ORGANIZATION_BLOCK "COMPLETE RESTART"
TITLE =Force glue-scale / Panel LED state to safe idle on every PLC restart
// v0.1 - NEW, per Michou's request (2026-10-06): "need to reset
//   everything when PLC reboots." S7-300 DB "actual values" are
//   battery/cap-backed and survive a power cycle - without this, a
//   reboot mid-recalibration would leave ReCalib_Step stuck mid-sequence
//   while K1/K2 are physically de-energized (CPU zeroes the output
//   process image on every restart, before this OB even runs), and any
//   latched alarms or Panel LED test bits would resume as if nothing
//   happened. Networks below force this repo's own state fields back to
//   a safe idle/off default. Operator setpoints (Fill_Start_SP,
//   Fill_Stop_SP, AlarmLimit_*_SP, PlatformMinWeight_SP,
//   NegativeUnderScore_Value) are deliberately NOT touched here - those
//   are calibration, not state, and must survive a reboot.
//
//   IMPORTANT, CONFIRMED (Michou, 2026-10-06): OB100 already exists on
//   the live PLC project. Michou - paste this file's networks into the
//   END of your existing OB100, do NOT download/replace the whole
//   block - that would silently delete whatever else it already resets
//   for other 410 subsystems. This tracked file only ever represents
//   the networks this repo's own subsystems need, not the real OB100.
//
// v0.2 - per Michou (2026-10-06): "Need a 30 sec delay before
//   restarting after power has resumed ... Need to restart KiloTech
//   Scale too and make sure it is calibrated before operating the
//   pump!" OB100 itself can't block/delay (an OB can't sit and wait -
//   that would trip the scan-time watchdog) - the actual 30s wait and
//   auto-recalibration run in FC155/FB555 (v0.30/v0.4), gated by two
//   new DB105 bits this OB resets every restart: PowerUp_Settled
//   (drives FB555's new 30s startup timer - see FC155's "Timers"
//   network) and Scale_Calibrated (the new pump interlock - see FC155's
//   "Power-up/recalibration interlock" network). Added both resets to
//   the "Glue scale" network below.
//
// v0.3 - reconciled against Michou's own live DB105 refactor
//   (2026-10-07): Reset_Alarms renamed Alarms_Acknowledge - updated the
//   reset below to match. Also added a reset for the new
//   Alarm_PossibleLeak latch (FC155/DB105 v0.20) - missed when that
//   alarm was first added, would have left a possible-leak alarm from
//   before a reboot still latched after it.
VERSION : 0.3


VAR_TEMP
  OB100_EV_CLASS : BYTE ;
  OB100_STRTUP : BYTE ;
  OB100_PRIORITY : BYTE ;
  OB100_OB_NUMBR : BYTE ;
  OB100_RESERVED_1 : BYTE ;
  OB100_RESERVED_2 : BYTE ;
  OB100_STOP : WORD ;
  OB100_STRT_INFO : DWORD ;
  OB100_DATE_TIME : DATE_AND_TIME ;
END_VAR
BEGIN
NETWORK
TITLE =Glue scale - clear latched alarms, HMI trigger pulses, and mid-sequence state (see FC155)

      R     "GLUE SCALE CONTROL DB".Pump_ON;
      R     "GLUE SCALE CONTROL DB".Alarm_Overfill;
      R     "GLUE SCALE CONTROL DB".Alarm_Underfill;
      R     "GLUE SCALE CONTROL DB".Alarm_ScaleFault;
      R     "GLUE SCALE CONTROL DB".ParseError;
      R     "GLUE SCALE CONTROL DB".Pump_ON_Prev;
      R     "GLUE SCALE CONTROL DB".Scale_Powered_On;
      R     "GLUE SCALE CONTROL DB".Alarms_Acknowledge;
      R     "GLUE SCALE CONTROL DB".Alarm_PossibleLeak;
      R     "GLUE SCALE CONTROL DB".Scale_PowerOFF_Pulse;
      R     "GLUE SCALE CONTROL DB".Scale_ReCalib_Req;
      R     "GLUE SCALE CONTROL DB".Scale_PowerON_Pulse;
      R     "GLUE SCALE CONTROL DB".LampScanClockMem;
      R     "GLUE SCALE CONTROL DB".PowerUp_Settled;
      R     "GLUE SCALE CONTROL DB".Scale_Calibrated;

      L     0;
      T     "GLUE SCALE CONTROL DB".ReCalib_Step;
      L     1;
      T     "GLUE SCALE CONTROL DB".LampScanStep;
      L     -20663;
      T     "GLUE SCALE CONTROL DB".GrossWeight_Actual;
      L     0;
      T     "GLUE SCALE CONTROL DB".GrossWeight_Actual_Mem;
      L     0;
      T     "GLUE SCALE CONTROL DB".Actual_Transfered_Weight;

NETWORK
TITLE =KILOTECK relays - force off explicitly (belt-and-suspenders; the CPU already zeroes physical outputs on restart)

      R     "OUTPUTS DB".KILOTECK_Calib_K1;
      R     "OUTPUTS DB".KILOTECK_Power_K2;

NETWORK
TITLE =Panel LED command bits - force idle, see FC157/DB107 (any caller must re-request behavior after a reboot)

      R     "PANEL LED CMD DB".WHT_ScanFwd;
      R     "PANEL LED CMD DB".WHT_ScanRev;
      R     "PANEL LED CMD DB".WHT_Panic;
      R     "PANEL LED CMD DB".WHT_1;
      R     "PANEL LED CMD DB".WHT_2;
      R     "PANEL LED CMD DB".WHT_3;
      R     "PANEL LED CMD DB".GRN_On;
      R     "PANEL LED CMD DB".GRN_Blink;
      R     "PANEL LED CMD DB".RED_On;
      R     "PANEL LED CMD DB".RED_Blink;

      L     1;
      T     "PANEL LED CMD DB".WHT_ScanStep;

END_ORGANIZATION_BLOCK
